{attribute 'qualified_only'}
//{attribute 'strict'}
{attribute 'to_string'}
TYPE E_NCI_STATE :
(
  NO_NCI            := -10,
  NO_AXIS_GROUP     := -2,
  NO_AXIS_INDEX     := -1,
  NO_INIT,
  INIT,
  IDLE,
  RESET,
  LOAD_PROG,
  FEED_TABLE,
  BUILD_GROUP,
  CLEAR_GROUP,

  START         := 10,
  STOP,
  STO_STOP,
  RESTART_STEP_ON,

  M_FUNC_QUIT   := 20,

  READ_R_PARA   := 30,
  WRITE_R_PARA  := 40

)DINT;
END_TYPE

(* stored: Version 1.1.0.1, ProductVersion 3.1.4024.12
   DUT E_NCI_STATE: Id {2b055dfa-b4d9-043d-259a-9033afd60d84} *)
